RoboDK station: Assistive_UR5e.rdk

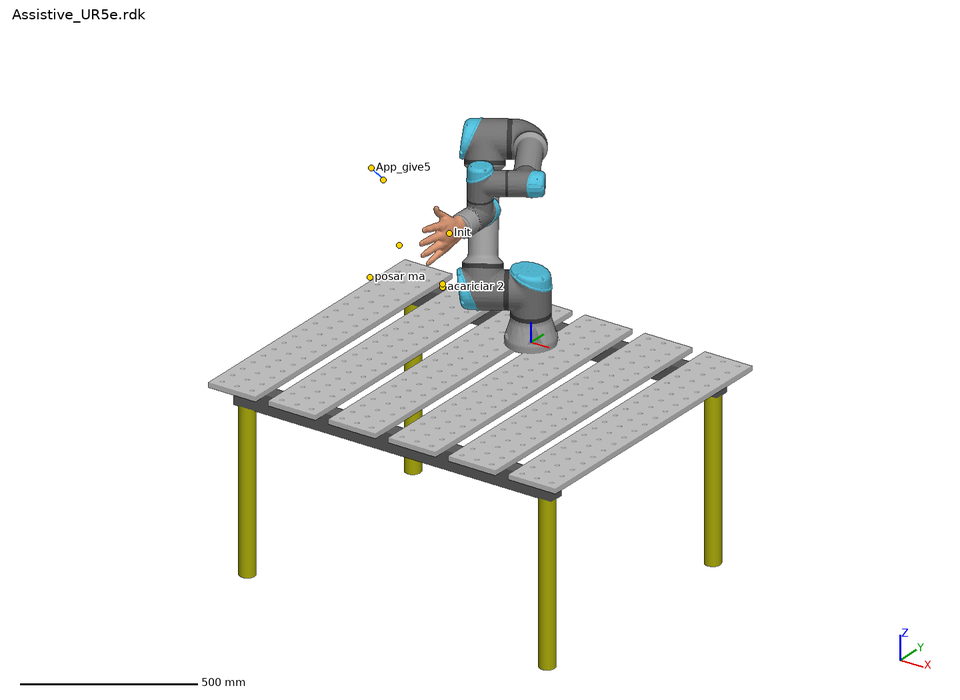
[picture v0: the station drawn from its stored meshes, robots at their saved joint values, targets as dots, program paths as lines]
Station Assistive_UR5e_SW (saved by RoboDK 5.9.2). Poses are relative to the parent item; angles as X-Y-Z fixed-axis rotations.
  - frame UR5e Base at (0, 0, 0) mm
    - robot UR5e: 6 axes, payload 5 kg, reach 850 mm, repeatability 0.03 mm, weight 18.4 kg
        modified DH rows (alpha deg, a mm, theta deg, d mm): 0, 0, 0, 162.5; 90, 0, 180, 0; 0, 425, 0, 0; 0, 392.25, 0, 133.3; -90, 0, 0, 99.7; 90, 0, 180, 99.6
        joint limits [-360, -360, -360, -360, -360, -360] to [360, 360, 360, 360, 360, 360]; home [0, -90, -90, 0, 90, 0]; saved at [-57.836, -65.392, -107.167, -187.441, -57.836, 0]
      - tool Hand, TCP at (0, 0, 50) mm, size 54.8 x 155.9 x 193.5 mm, geometry from Hand.stl
  - frame World at (0, 0, 0) mm
    - object Table at (0, 0, 0) mm, size 1193.8 x 965.2 x 609.6 mm, geometry from welding_table.sld
    - target Init (Cartesian target) at (0, -400, 500) mm, rotated rx 90 ry 0 rz 0 deg; joints [-57.836, -65.392, -107.167, -187.441, -57.836, 0] of UR5e
    - target posar ma (Cartesian target) at (-350, -290, 220) mm, rotated rx 45 ry 90 rz -45 deg; joints [-137.442, 146.423, -236.23, 89.807, 222.558, -90] of UR5e
    - target acariciar 1 (Cartesian target) at (-250, -290, 350) mm, rotated rx 90 ry -70 rz 0 deg; joints [-122.977, -73.689, -124.232, -162.079, -122.977, 70] of UR5e
    - target acariciar 2 (Cartesian target) at (-100, -290, 260) mm, rotated rx 90 ry -70 rz 0 deg; joints [3.886, 5.109, -148.295, -216.816, 3.886, 70.001] of UR5e
    - target acariciar 1 (Cartesian target) at (-250, -290, 350) mm, rotated rx 90 ry -70 rz 0 deg; joints [1.615, 9.258, -124.233, -245.03, 1.615, 70.004] of UR5e
    - target acariciar 2 (Cartesian target) at (-100, -290, 269) mm, rotated rx 90 ry -70 rz 0 deg; joints [-74.807, -52.096, -147.127, -160.778, -74.807, 69.999] of UR5e
    - target acariciar 1 (Cartesian target) at (-250, -290, 350) mm, rotated rx 90 ry -70 rz 0 deg; joints [-122.977, -73.689, -124.232, -162.079, -122.977, 70] of UR5e
    - target App_give5 (joint target) at (-380.86, -238.62, 533.82) mm, rotated rx 0 ry 0 rz 90 deg; joints [-130.679, -89.195, -122.013, 301.208, -90, 130.679] of UR5e
    - target HOLA 1 (joint target) at (-310.86, -280, 533.82) mm, rotated rx -30 ry 0 rz 90 deg; joints [-108.789, -73.555, -128.554, 281.574, -61.748, 111.447] of UR5e
    - target HOLA 2 (Cartesian target) at (-310.86, -280, 533.82) mm, rotated rx 30 ry 0 rz 90 deg; joints [-127.777, -94.791, -118.448, 322.716, -113.278, 131.827] of UR5e
  - program Init (3 instructions, listed below)
  - program Hand_shake (5 instructions, listed below)
  - program Give_me_5! (5 instructions, listed below)
  - program MainProgram (4 instructions, listed below)
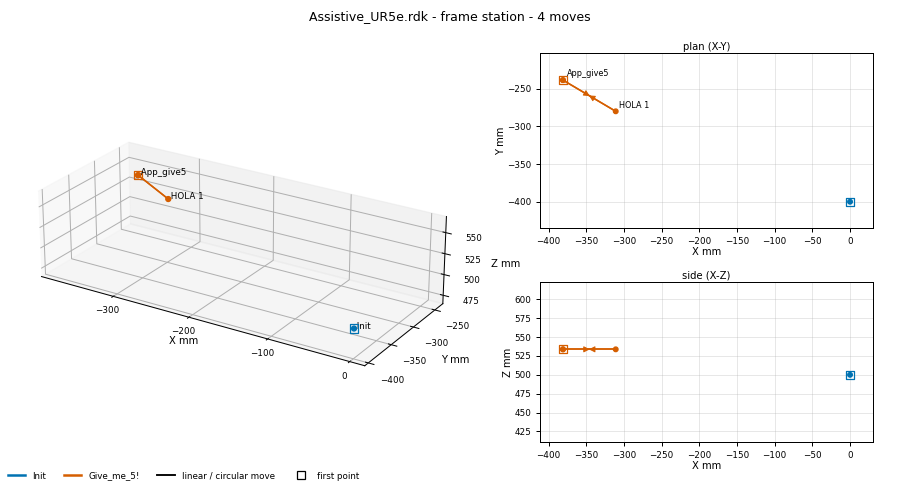
[picture p0: tool path of Assistive_UR5e.rdk in frame station, 4 of 7 moves have a stored position in this frame; points joined in program order, loops and branches not executed]

--- program Init (robot UR5e) ---
  Est. Ref.: UR5e Base
  Est. herr: Hand
  MoveJ (Init)

--- program Hand_shake (robot UR5e) ---
  Est. Ref.: UR5e Base
  Est. herr: Hand
  MoveL (App_shake) [its target is no longer in the station]
  MoveL (Shake) [its target is no longer in the station]
  MoveL (App_shake) [its target is no longer in the station]

--- program Give_me_5! (robot UR5e) ---
  Est. Ref.: UR5e Base
  Est. herr: Hand
  MoveL (App_give5)
  MoveL (Give5) -> target HOLA 1
  MoveL (App_give5)

--- program MainProgram (robot UR5e) ---
  Llamar Init
  Llamar Hand_shake
  Llamar Give_me_5!
  Llamar Init
